# B&R Automation Studio project lektion_9_agdp
Automation Studio 4.8.2.72

## Configuration Config1

### Task classes (Cpu.sw)
```
Cyclic#1:
  Assignmen1 <- Assignment2.prg
  Assignment <- Assignment1.prg
  Assignmen2 <- Assignment3.prg
Binaries: udbdef, FWRules, TCData, sysconf, Role, User, iomap, ashwd, asfw, arconfig, ashwac
Libraries: standard, runtime, astime, asieccon
```

### Hardware
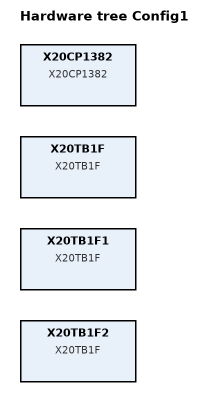
```
X20CP1382 : X20CP1382 v1.10.0.0  [X1 -> X1.SL; X2 -> X2.SL; X3 -> X3.SL]
  Module X1 (Type=X1, Virtual=true, Version=1.10.0.0)
    Connection (Connector=SS1, TargetModule=X20TB1F, TargetConnector=SS)
    Connection (Connector=SL, TargetModule=X20CP1382, TargetConnector=X1)
  Module X2 (Type=X2, Virtual=true, Version=1.10.0.0)
    Connection (Connector=SS1, TargetModule=X20TB1F1, TargetConnector=SS)
    Connection (Connector=SL, TargetModule=X20CP1382, TargetConnector=X2)
  Module X3 (Type=X3, Virtual=true, Version=1.10.0.0)
    Connection (Connector=SS1, TargetModule=X20TB1F2, TargetConnector=SS)
    Connection (Connector=SL, TargetModule=X20CP1382, TargetConnector=X3)
  Connector IF2:
    ActivateDevice = 1
  ConfigurationID = lektion_9_agdp_Config1
  Simulation = 1
X20TB1F : X20TB1F v1.0.0.0
X20TB1F1 : X20TB1F v1.0.0.0
X20TB1F2 : X20TB1F v1.0.0.0
```

## Logical view

### Program Logical/Assignment1 (IEC)

#### Main.st - Init, cyclic, exit code
```iecst
PROGRAM _INIT
	(* Insert code here *)

END_PROGRAM

PROGRAM _CYCLIC
	// Tilstandsskiftlogik / state change logic
	CASE castate OF
		CARALARM_DISARMED:
			IF diRemote AND flag THEN
				castate := CARALARM_ARMED;
			END_IF

		CARALARM_ARMED:
			IF diRemote AND flag THEN
				castate := CARALARM_DISARMED;
			ELSIF diSensorVibration THEN
				castate := CARALARM_INTRUSION;
			END_IF

		CARALARM_INTRUSION:
			IF diRemote AND flag THEN
				castate := CARALARM_DISARMED;
			END_IF
	END_CASE

	flag := NOT old_remote AND diRemote;
	old_remote := diRemote;

	// Output logic
	CASE castate OF
		CARALARM_DISARMED:
			doSiren := FALSE;

		CARALARM_ARMED:

		CARALARM_INTRUSION:
			doSiren := TRUE;
	END_CASE

END_PROGRAM

PROGRAM _EXIT
	(* Insert code here *)

END_PROGRAM
```

#### Types.typ - Local data types
```iecst
TYPE
	CARALARM :
		(
		CARALARM_DISARMED,
		CARALARM_ARMED,
		CARALARM_INTRUSION
		);
END_TYPE
```

#### Variables.var - Local variables
```iecst
VAR
	castate : CARALARM;
	diSensorVibration : BOOL;
	old_remote : BOOL;
	flag : BOOL;
	diRemote : BOOL;
	doSiren : BOOL;
END_VAR
```

### Program Logical/Assignment2 (IEC)

#### Types.typ
```iecst
TYPE
	TRAFFICLIGHT :
		(
		STOPPED,
		READY,
		STOP,
		GO
		);
END_TYPE
```

#### Variables.var
```iecst
VAR
	castate : TRAFFICLIGHT;
	yellow : BOOL;
	green : BOOL;
	red : BOOL;
	timer : TON;
END_VAR
```

#### Main.st
```iecst
PROGRAM _INIT
	(* Insert code here *)

END_PROGRAM

PROGRAM _CYCLIC
	// Tilstandsskiftlogik / state change logic
	timer.IN := TRUE;
	CASE castate OF
		STOPPED:
			timer.PT := T#5s;
			IF timer.Q THEN
				castate := READY;
				timer.IN := FALSE;
			END_IF;
		READY:
			timer.PT := T#3s;
			IF timer.Q THEN
				castate := GO;
				timer.IN := FALSE;
			END_IF;
		GO:
			timer.PT := T#7s;
			IF timer.Q THEN
				castate := STOP;
				timer.IN := FALSE;
			END_IF;
		STOP:
			timer.PT := T#3s;
			IF timer.Q THEN
				castate := STOPPED;
				timer.IN := FALSE;
			END_IF;
	END_CASE
	timer();

	// OUTPUT LOGIC
	CASE castate OF
		STOPPED:
			yellow := FALSE;
			red := TRUE;
		READY:
			yellow := TRUE;
		GO:
			red := FALSE;
			yellow := FALSE;
			green := TRUE;
		STOP:
			yellow := TRUE;
			green := FALSE;

	END_CASE
END_PROGRAM

PROGRAM _EXIT
	(* Insert code here *)

END_PROGRAM
```

### Program Logical/Assignment3 (IEC)

#### Types.typ
```iecst
TYPE
	BLINDS :
		(
		OPEN,
		OPENING,
		CLOSED,
		CLOSING
		);
END_TYPE
```

#### Variables.var
```iecst
VAR
	castate : BLINDS;
	diOpen : BOOL;
	diClose : BOOL;
	timer : TON;
	doMoveDown : BOOL;
	doMoveUp : BOOL;
END_VAR
```

#### Main.st
```iecst
PROGRAM _INIT
	(* Insert code here *)
	timer.IN := FALSE;
END_PROGRAM

PROGRAM _CYCLIC
	// Tilstandsskiftlogik / state change logic
	// "di" stands for digital input.
	CASE castate OF
		OPEN:
			timer.IN := FALSE;
			IF diClose THEN
	  			castate := CLOSING;
			END_IF;
		CLOSING:
			timer.IN := TRUE;
			timer.PT := T#5s;
			IF timer.Q THEN
				castate := CLOSED;
			END_IF;
		CLOSED:
			timer.IN := FALSE;
			IF diOpen THEN
				castate := OPENING;
			END_IF;
		OPENING:
			timer.IN := TRUE;
			timer.PT := T#6s;
			IF timer.Q THEN
				castate := OPEN;
			END_IF;

	END_CASE
	timer();

	// OUTPUT LOGIC
	// "do" stands for digital output.
	CASE castate OF
		OPEN:
			doMoveUp := FALSE;
			doMoveDown := FALSE;
		CLOSING:
			doMoveUp := FALSE;
			doMoveDown := TRUE;
		CLOSED:
			doMoveUp := FALSE;
			doMoveDown := FALSE;
		OPENING:
			doMoveUp := TRUE;
			doMoveDown := FALSE;

	END_CASE
END_PROGRAM

PROGRAM _EXIT
	(* Insert code here *)

END_PROGRAM
```

Listed in the project but not available here: Logical/Global.typ, Logical/Global.var, Logical/Libraries
